{attribute addProperty BoxType "EK1960-0000-0019"}
{attribute addProperty Id "Module_1_FSoEModule_1_FSoE_DD00D81F240300Module_2_FSOUTModule_2_FSOUT_3AD10D8E224280Module_3_FSLOGICModule_3_FSLOGIC_3E6251391620WcStateAT %I*WcState_C1B70B0F3240InfoDataAT %I*InfoData_BC63D37F80100"}
{attribute addProperty CRC "4171187034"}
{attribute addProperty SizeInBites "592"}
{attribute addProperty SizeInBytes "74"}
TYPE EK1960_19ACB9CA :
STRUCT
	{attribute addProperty Name "Module_1_FSoE"}
	Module_1_FSoE : Module_1_FSoE_DD00D81F;
	{attribute addProperty Name "Module_2_FSOUT"}
	Module_2_FSOUT : Module_2_FSOUT_3AD10D8E;
	{attribute addProperty Name "Module_3_FSLOGIC"}
	Module_3_FSLOGIC : Module_3_FSLOGIC_3E625139;
	{attribute addProperty Name "WcState"}
	WcState : WcState_C1B70B0F;
	{attribute addProperty Name "InfoData"}
	InfoData : InfoData_BC63D37F;
END_STRUCT
END_TYPE

(* stored: Version 1.2.0.0, ProductVersion 3.1.4024.9
   DUT EK1960_19ACB9CA: Id {b6d2c563-4d44-4021-a4ae-5ebcd120f81d} *)
